(* PLC project KinIn_v3.project, CODESYS CODESYS V3.5 SP19 *)
(* stored: creationDateTime 2025-01-20T16:28:35.4990452, modificationDateTime 2025-01-20T16:17:39.6822999 *)

FUNCTION_BLOCK INV_KINEMATICS
  VAR_INPUT
    M : ARRAY[1..4, 1..4] OF REAL;
    T : ARRAY[1..4, 1..4] OF REAL;
    eomg : REAL;
    ev : REAL;
    nIterationsIK : DINT;
    Blist : ARRAY[1..6, 1..GVL.nJoints] OF REAL;
  END_VAR
  VAR_OUTPUT
    thetalist : ARRAY[1..GVL.nJoints] OF REAL;  (* as output *)
    q_IKsuccess : BOOL;
    s_IK_message : STRING;
  END_VAR
  VAR
    RndStart : RndStart;
    getInvKinematics_Body : getInvKinematics_Body;
    success : BOOL;
    i_iteration : DINT;
    q_JointOK : BOOL;
    thetalist0 : ARRAY[1..GVL.nJoints] OF REAL;
    i : DINT;
  END_VAR

            	(*-----------for various iterations of IK---------*)
//random start with compliant joint limits
i_iteration:=0;q_IKsuccess:=FALSE;
WHILE (i_iteration<nIterationsIK	 AND  q_IKsuccess=FALSE) DO
	RndStart(ar_JointLimits:=GVL.ar_JointLimits , randomArray=>thetalist0 );	
	
	getInvKinematics_Body(
		M:=M , 
		T:=T , 
		eomg:= eomg, 
		ev:= ev, 
		Blist:=Blist , 
		thetalist0:= thetalist0, 
		thetalist:=thetalist , 
		success=> success);	
	
	i:=1;q_JointOK:=TRUE;q_IKsuccess:=TRUE;
	FOR i:=1 TO UPPER_BOUND(thetalist,1) DO	
		q_JointOK:=GVL.ar_JointLimits[i,1]<=thetalist[i] AND thetalist[i]<=GVL.ar_JointLimits[i,2];
		IF q_JointOK=FALSE THEN
			q_IKsuccess:=FALSE;
		END_IF
	END_FOR
	i_iteration:=i_iteration+1;
END_WHILE

IF (i_iteration>=nIterationsIK	 AND  q_IKsuccess=FALSE) THEN
	s_IK_message:='Could not solve the inverse kinematics';
ELSE
	s_IK_message:='The inverse kinematics was completed';
END_IF
          
END_FUNCTION_BLOCK
